INTERFACE I_CollisionGroup

METHOD AddMoverToThisGroup : HRESULT
VAR_INPUT
	MoverToAdd : I_XtsMover;
END_VAR
END_METHOD

PROPERTY AxisCount : UDINT
GET
END_GET
END_PROPERTY

PROPERTY CAGroupXtsIoEnvInterface : I_Mc2CaGroup
GET
END_GET
SET
END_SET
END_PROPERTY

METHOD Disable : BOOL
VAR_INPUT
END_VAR
END_METHOD

METHOD Enable : BOOL
VAR_INPUT
END_VAR
END_METHOD

PROPERTY ErrorCode : UDINT
GET
END_GET
END_PROPERTY

PROPERTY GroupRef : reference to AXES_GROUP_REF
GET
END_GET
END_PROPERTY

METHOD GroupStop : BOOL
VAR_INPUT
END_VAR
END_METHOD

PROPERTY HasError : BOOL
GET
END_GET
END_PROPERTY

PROPERTY IsDisabled : BOOL
GET
END_GET
END_PROPERTY

PROPERTY IsInErrorStop : BOOL
GET
END_GET
END_PROPERTY

PROPERTY IsInStandBy : BOOL
GET
END_GET
END_PROPERTY

PROPERTY IsMoving : BOOL
GET
END_GET
END_PROPERTY

PROPERTY IsStopping : BOOL
GET
END_GET
END_PROPERTY

PROPERTY MyName : string
GET
END_GET
END_PROPERTY

METHOD RemoveAllMovers : HRESULT
VAR_INPUT
END_VAR
END_METHOD

METHOD RemoveAMover : HRESULT
VAR_INPUT
	MoverToRemove : I_XtsMover;
END_VAR
END_METHOD

METHOD Reset : HRESULT
VAR_INPUT
END_VAR
END_METHOD

END_INTERFACE

(* stored: Version 1.1.0.1
   Itf I_CollisionGroup: Id {3fc566cf-3f15-4187-97a8-f8d156c2ea05}
   Folder Commands: Id {8beee7c9-6c57-495f-8157-bb3d16e9e090}
   Folder Status: Id {c894277c-e5b7-477b-b238-fbc580fc1f1e}
   Method AddMoverToThisGroup: Id {e0521e35-3414-4dd6-b2e7-4ac92ca8a051}
   Property AxisCount: Id {a5c90290-77cc-4f48-9b6f-5a9162b91e28}
   Get Get: Id {ea8e9e75-8d55-40e9-a8b8-94e9484ee31a}
   Property CAGroupXtsIoEnvInterface: Id {cd5d9462-f9cf-4d35-b22c-6eae8c9cec38}
   Get Get: Id {4b7a5dbd-2b80-4c96-b418-833e5507e708}
   Set Set: Id {a85ceeb9-ae20-4fa6-83c9-e0f32834f786}
   Method Disable: Id {716927af-8c3f-479d-962f-20b060f08214}
   Method Enable: Id {7961c446-8ffb-4a93-bee2-efac793ad03b}
   Property ErrorCode: Id {45e0d2f7-1cdd-4165-ae7f-f50369fa11b7}
   Get Get: Id {e1e19d43-f378-460b-b455-9c54804e6dfd}
   Property GroupRef: Id {da70f768-e857-4f18-9014-1c57ab869df0}
   Get Get: Id {ff65d9fd-a0fb-4014-a5bd-11ea974f60f4}
   Method GroupStop: Id {da0fa42b-dbcd-4e72-85b3-93d42f55308f}
   Property HasError: Id {557f11a2-aaf0-4723-830e-c7d87858b60f}
   Get Get: Id {ba4be547-d47a-41bc-9b1a-df5c5f0deff3}
   Property IsDisabled: Id {d615efc1-92df-43ae-9bd1-e7a398601ddf}
   Get Get: Id {bc9ef1c8-c7b5-444d-ae03-89d190539ae0}
   Property IsInErrorStop: Id {5023391e-44dd-406b-b3b5-f9ea9ac32b34}
   Get Get: Id {3e12ed68-1f99-4bf5-b7b0-15da1afa0b14}
   Property IsInStandBy: Id {c30e3728-c4be-4b2b-8e19-f5d930f52e82}
   Get Get: Id {18e6e8d8-2be4-4163-ab4e-ba882d459ce9}
   Property IsMoving: Id {ab17e853-c3bd-4d23-afdc-251dc4495b75}
   Get Get: Id {5039bbf0-2360-4c71-8dd2-01ca1383f74d}
   Property IsStopping: Id {1421d697-4b12-474e-9928-b9a704264869}
   Get Get: Id {22fd8dae-d519-4985-b0ce-cc050c1bc3e4}
   Property MyName: Id {989d2fa8-4a9f-4077-ad60-57e1e6700080}
   Get Get: Id {962bda42-6307-4da5-99e1-648fbb7790b1}
   Method RemoveAllMovers: Id {ef3d94da-4e03-448c-b177-7286a6d747e3}
   Method RemoveAMover: Id {ef48cf2e-8bac-48d4-bde6-7be9e9dfb88f}
   Method Reset: Id {52cfbceb-29c1-48af-b76e-6022383fab33} *)
